// Mitsubishi GX Works2 project: 0702-행님답지   PLC: Q02/Q02H

PROGRAM MAIN
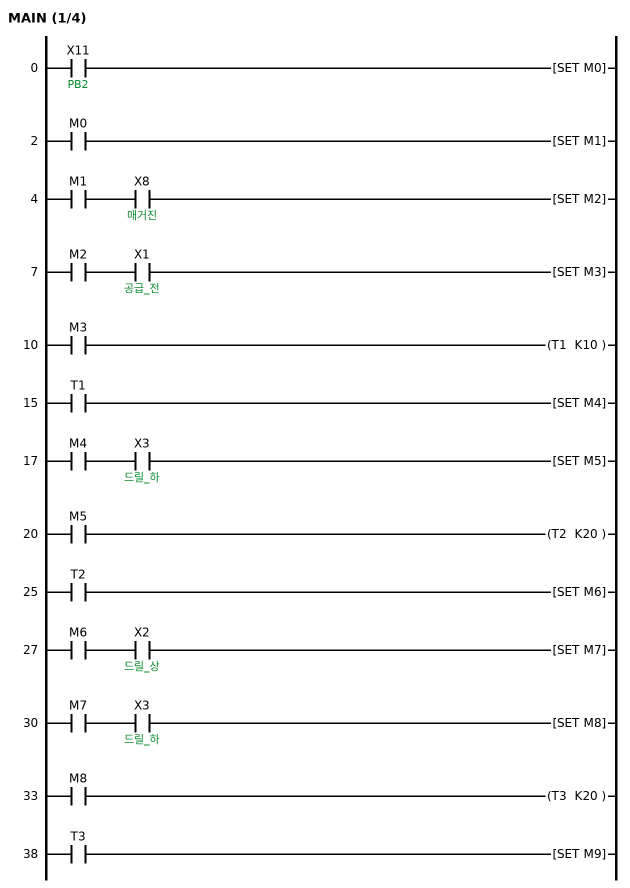
0     LD      X11  ; PB2
      SET     M0
2     LD      M0
      SET     M1
4     LD      M1
      AND     X8  ; 매거진
      SET     M2
7     LD      M2
      AND     X1  ; 공급_전
      SET     M3
10    LD      M3
      OUT     T1 K10
15    LD      T1
      SET     M4
17    LD      M4
      AND     X3  ; 드릴_하
      SET     M5
20    LD      M5
      OUT     T2 K20
25    LD      T2
      SET     M6
27    LD      M6
      AND     X2  ; 드릴_상
      SET     M7
30    LD      M7
      AND     X3  ; 드릴_하
      SET     M8
33    LD      M8
      OUT     T3 K20
38    LD      T3
      SET     M9
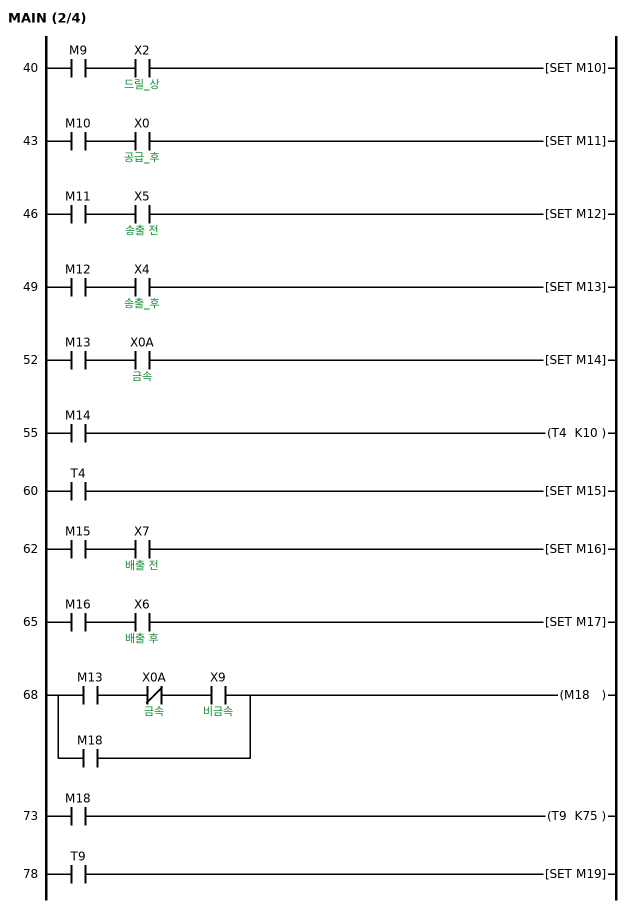
40    LD      M9
      AND     X2  ; 드릴_상
      SET     M10
43    LD      M10
      AND     X0  ; 공급_후
      SET     M11
46    LD      M11
      AND     X5  ; 송출 전
      SET     M12
49    LD      M12
      AND     X4  ; 송출_후
      SET     M13
52    LD      M13
      AND     X0A  ; 금속
      SET     M14
55    LD      M14
      OUT     T4 K10
60    LD      T4
      SET     M15
62    LD      M15
      AND     X7  ; 배출 전
      SET     M16
65    LD      M16
      AND     X6  ; 배출 후
      SET     M17
68    LD      M13
      ANI     X0A  ; 금속
      AND     X9  ; 비금속
      OR      M18
      OUT     M18
73    LD      M18
      OUT     T9 K75
78    LD      T9
      SET     M19
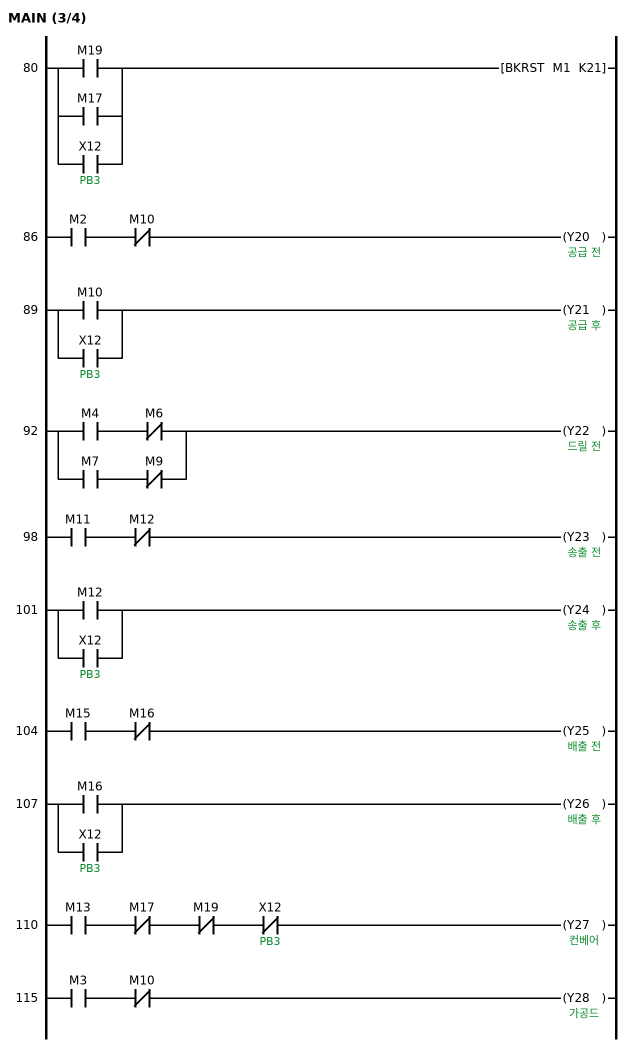
80    LD      M19
      OR      M17
      OR      X12  ; PB3
      BKRST   M1 K21
86    LD      M2
      ANI     M10
      OUT     Y20  ; 공급 전
89    LD      M10
      OR      X12  ; PB3
      OUT     Y21  ; 공급 후
92    LD      M4
      ANI     M6
      LD      M7
      ANI     M9
      ORB
      OUT     Y22  ; 드릴 전
98    LD      M11
      ANI     M12
      OUT     Y23  ; 송출 전
101   LD      M12
      OR      X12  ; PB3
      OUT     Y24  ; 송출 후
104   LD      M15
      ANI     M16
      OUT     Y25  ; 배출 전
107   LD      M16
      OR      X12  ; PB3
      OUT     Y26  ; 배출 후
110   LD      M13
      ANI     M17
      ANI     M19
      ANI     X12  ; PB3
      OUT     Y27  ; 컨베어
115   LD      M3
      ANI     M10
      OUT     Y28  ; 가공드
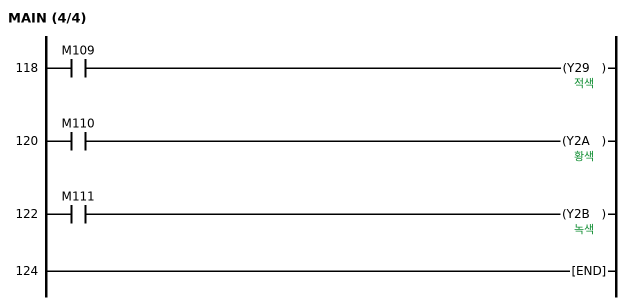
118   LD      M109
      OUT     Y29  ; 적색
120   LD      M110
      OUT     Y2A  ; 황색
122   LD      M111
      OUT     Y2B  ; 녹색
124   END
END_PROGRAM

// device comments not shown above
X10  ; PB1
